FUNCTION_BLOCK T_RoboConnect_SetToolDigitalOutput_IncorrectIndexFails EXTENDS T_UnitTestBase
VAR
  robot : I_RoboConnect;
  targetDO : UINT;
  myTestState, prevState :
    (INIT, ARRANGE, ACT, ASSERT)
    := INIT;
  expected : BOOL;
  actual : BOOL := TRUE;
  counter : UINT;
END_VAR

CASE myTestState OF
  INIT:
    StateChanged();
    myTestState := ARRANGE;

  ARRANGE:
    IF StateChanged() THEN
      expected := FALSE;
      myTestState := ACT;
    END_IF

  ACT:
    actual := robot.SetToolDigitalOutput(targetDO, TRUE);
    myTestState := ASSERT;

  ASSERT:
    assertion.AssertEquals_BOOL(expected, actual, 'robot.GetDigitalOutput(targetDO) := TRUE');
    TestFinished();
    myTestState := INIT;

END_CASE

METHOD FB_init : BOOL
VAR_INPUT
  bInitRetains : BOOL; // if TRUE, the retain variables are initialized (warm start / cold start)
  bInCopyCode : BOOL; // if TRUE, the instance afterwards gets moved into the copy code (online change)
  TestSuite : tcl_SimpleUnitTestLibrary.I_TestSuite;
  robot : I_TcRobot;
  targetDo : UINT;
END_VAR
THIS^.robot := robot;
THIS^.targetDo := targetDo;
END_METHOD

METHOD PRIVATE StateChanged : BOOL
IF  myTestState = prevState THEN
  RETURN;
END_IF

prevState := myTestState;
StateChanged := TRUE;
END_METHOD

METHOD WaitForCycles : BOOL
VAR_INPUT
  maxCount : UINT;
END_VAR
counter := counter + 1;

IF counter = maxCount THEN
  counter := 0;
  WaitForCycles := TRUE;
END_IF
END_METHOD

END_FUNCTION_BLOCK

(* stored: Version 1.1.0.1
   POU T_TcRobot_SetToolDigitalOutput_IncorrectIndexFails: Id {26962d04-05ef-4725-9b84-6b07bb54d80f}, SpecialFunc None
   Method FB_init: Id {613e5ab9-6c5f-46f8-bca2-dbfb621c9187}
   Method StateChanged: Id {41f52935-159a-44c3-b5e4-9965c9757d9f}
   Method WaitForCycles: Id {8ab28cd8-dcf5-43a5-9b5e-140af56433c5} *)
